FUNCTION_BLOCK ComparisonFunctionsTest EXTENDS TcUnit.FB_TestSuite
VAR
END_VAR

DataEqualsFunction();

METHOD DataEqualsFunction : BOOL
VAR
	data1 : INT;
	data2 : INT;
END_VAR
TcUnit.TEST('Data equals');

data1 := 42;
data2 := 0;

AssertEquals_BOOL(
	Expected := FALSE,
	Actual := DataEquals(data1, data2),
	Message := 'Data should not be equal');

data2 := data1;

AssertEquals_BOOL(
	Expected := TRUE,
	Actual := DataEquals(data1, data2),
	Message := 'Data should be equal');

TEST_FINISHED();
END_METHOD

END_FUNCTION_BLOCK

(* stored: Version 1.1.0.1, ProductVersion 3.1.4024.12
   POU ComparisonFunctionsTest: Id {f90bffaf-3a64-090c-126d-223f1ba9034f}, SpecialFunc None
   Method DataEqualsFunction: Id {6d0ce20e-9b64-0d8d-0ae4-3f5ee07fa4d9} *)
